// TIA Portal V20 export
FUNCTION "Bit_To_Word" : Void   // FC2, LAD
{ S7_Optimized_Access := 'TRUE' }
// stored: SetENOAutomatically false
   VAR_INPUT
      BIT : "UDT_Flowmeter_Stoe";
   END_VAR
   VAR_OUTPUT
      Out_I : Int;
   END_VAR
   VAR_TEMP
      Out_W : Word;
   END_VAR
BEGIN

REGION Network 1 (SCL)
   #Out_W :=0;

   IF #BIT."No Flow Detected" THEN
       #Out_W := #Out_W OR W#16#1;
   END_IF;

   IF #BIT."Flow Rate Too Low" THEN
       #Out_W := #Out_W OR W#16#2;
   END_IF;

   IF #BIT."Flow Rate Too Hight" THEN
       #Out_W := #Out_W OR W#16#4;
   END_IF;

   IF #BIT."Sensor CH1_wBreak" THEN
       #Out_W := #Out_W OR W#16#8;
   END_IF;

   IF #BIT."Sensor CH2_wBreak" THEN
       #Out_W := #Out_W OR W#16#10;
   END_IF;

   IF #BIT."Temprature Above Limit" THEN
       #Out_W := #Out_W OR W#16#20;
   END_IF;

   IF #BIT."Flow Out Of Range" THEN
       #Out_W := #Out_W OR W#16#40;
   END_IF;

   IF #BIT."Calibration Error" THEN
       #Out_W := #Out_W OR W#16#80;
   END_IF;

   IF   #BIT."Air Bubles Detected"    THEN
       #Out_W := #Out_W OR W#16#100;
   END_IF;

   IF #BIT."Temprature Out Of Range" THEN
       #Out_W := #Out_W OR W#16#200;
   END_IF;

   IF #BIT."Temprature Below Limit" THEN
       #Out_W := #Out_W OR W#16#400;
   END_IF;

   IF #BIT."Reverse Flow Detected" THEN
       #Out_W := #Out_W OR W#16#800;
   END_IF;

   IF #BIT."Communcation Error" THEN
       #Out_W := #Out_W OR W#16#1000;
   END_IF;

   IF #BIT."Clogging or Blockage" THEN
       #Out_W := #Out_W OR W#16#2000;
   END_IF;

   IF #BIT."Sensor Overheating" THEN
       #Out_W := #Out_W OR W#16#4000;
   END_IF;

   IF #BIT."Dirty Sensor" THEN
       #Out_W := #Out_W OR W#16#8000;
   END_IF;

   #Out_I := WORD_TO_INT(#Out_W);
END_REGION
END_FUNCTION
